(* Logix 5000 project; controller WWTP_SOLIDS_CLX vendor 1 type 14 code 54 rev 17.2; software revision 17.00; part 14 of 16 *)
(* tags used below, declared in another part *)
   Inp_ClosedLS : BOOL;   // Valve Closed Limit Switch 1=confirmed CLOSED
   Inp_OpenPermOK : BOOL;   // 1=Open Permissives OK, Valve can motor open
   Inp_OpenNBPermOK : BOOL;   // 1=Non-Bypassable Open Permissives OK, valve can motor open
   Inp_ClosePermOK : BOOL;   // 1=Close Permissives OK, Valve can motor closed
   Inp_CloseNBPermOK : BOOL;   // 1=Non-Bypassable Close Permissives OK, valve can motor closed
   Inp_IOFault : BOOL;   // Input Communication Status 0=OK, 1=fail
   Inp_Sim : BOOL;   // 1=Simulate working valve; 0=Open/Close/ Monitor actual valve
   Inp_Hand : BOOL;   // 1=Select Hand (hardwired) Mode
   Inp_Reset : BOOL;   // 1=Reset all fault conditions and latched Alarms
   Cfg_HasOpenLS : BOOL;   // 1=Valve provides an Open Limit Switch signal
   Cfg_HasClosedLS : BOOL;   // 1=Valve provides a Closed Limit Switch signal
   Cfg_UseOpenLS : BOOL;   // 1=Valve Open LS should be used for failure checking
   Cfg_UseClosedLS : BOOL;   // 1=Valve Closed LS should be used for failure checking
   Cfg_LSFail : BOOL;   // 1=both switches ON=fail, 0=both switches OFF=fail
   Cfg_HasOpenPermObj : BOOL;   // 1=Tells HMI a P_Perm is connected to Inp_OpenPermOK
   Cfg_HasClosePermObj : BOOL;   // 1=Tells HMI a P_Perm is connected to Inp_ClosePermOK
   Cfg_PCmdClear : BOOL;   // 1=Clear Program Commands on receipt 0=Leave Set
   Cfg_HasFullStallAlm : BOOL;   // 1=Full Stall Alarm exists and will be checked
   Cfg_HasTransitStallAlm : BOOL;   // 1=Transit Stall Alarm exists and will be checked
   Cfg_HasActuatorFaultAlm : BOOL;   // 1=Actuator Fault Alarm exists and will be checked
   Cfg_HasIOFaultAlm : BOOL;   // 1=I/O Fault Alarm exists and will be checked
   Cfg_FullStallAckReqd : BOOL;   // 1=Acknowledge required for Full Stall Alarm
   Cfg_TransitStallAckReqd : BOOL;   // 1=Acknowledge required for Transit Stall Alarm
   Cfg_ActuatorFaultAckReqd : BOOL;   // 1=Acknowledge required for Actuator Fault Alarm
   Cfg_IOFaultAckReqd : BOOL;   // 1=Acknowledge required for I/O Fault Alarm
   Cfg_FullStallSeverity : SINT;   // Full Stall Alarm Severity 1=info 2=warn 3=excep 4=fault
   Cfg_TransitStallSeverity : SINT;   // Transit Stall Alarm Severity 1=info 2=warn 3=excep 4=fault
   Cfg_ActuatorFaultSeverity : SINT;   // Actuator Fault Alarm Severity 1=info 2=warn 3=excep 4=fault
   Cfg_IOFaultSeverity : SINT;   // I/O Fault Alarm Severity 1=info 2=warn 3=excep 4=fault
   Cfg_OutPulseT : DINT;   // Time (in seconds) to pulse valve outputs (0 = outputs maintained ON)
   Cfg_SimFdbkT : DINT;   // Delay to echo back of Open/Closed status when in Simulation (sec)
   Cfg_FullStallT : DINT;   // After commanded, time with no motion before Fault (sec)
   Cfg_TransitStallT : DINT;   // After command, time to reach position before fault (sec)
   PSet_Owner : DINT;   // Program Owner Request ID (non-zero) or Release (zero)
   PCmd_Open : BOOL;   // Program Command to Open Valve
   PCmd_Close : BOOL;   // Program Command to Close Valve
   PCmd_Acq : BOOL;   // Program Command to Acquire ownership (Oper/OOS to Prog)
   PCmd_Rel : BOOL;   // Program Command to Release ownership (Prog to OOS)
   PCmd_Lock : BOOL;   // Program Command to Lock Mode in Prog
   PCmd_Unlock : BOOL;   // Program Command to Unlock Mode
   PCmd_Reset : BOOL;   // Program Command to Reset all Alarms requiring Reset
   PCmd_FullStallInhibit : BOOL;   // Program Command to Inhibit Full Stall Alarm
   PCmd_FullStallUninhibit : BOOL;   // Program Command to Uninhibit Full Stall Alarm
   PCmd_TransitStallInhibit : BOOL;   // Program Command to Inhibit Transit Stall Alarm
   PCmd_TransitStallUninhibit : BOOL;   // Program Command to Uninhibit Transit Stall Alarm
   PCmd_ActuatorFaultInhibit : BOOL;   // Program Command to Inhibit Actuator Fault Alarm
   PCmd_ActuatorFaultUninhibit : BOOL;   // Program Command to Uninhibit Actuator Fault Alarm
   PCmd_IOFaultInhibit : BOOL;   // Program Command to Inhibit I/O Fault Alarm
   PCmd_IOFaultUninhibit : BOOL;   // Program Command to Uninhibit I/O Fault Alarm
   OCmd_Open : BOOL;   // Operator Command to Open Valve
   OCmd_Close : BOOL;   // Operator Command to Close Valve
   OCmd_Stop : BOOL;   // Operator Command to Stop Valve Motion
   OCmd_Bypass : BOOL;   // Operator Command to Bypass all Bypassable Interlocks and Permissives
   OCmd_Check : BOOL;   // Operator Command to Check (not bypass) all Interlocks and Permissives
   MCmd_Disable : BOOL;   // Maintenance Command to Disable Valve
   MCmd_Enable : BOOL;   // Maintenance Command to Enable (allow to energize) Valve
   OCmd_Reset : BOOL;   // Operator Command to Reset all Alarms requiring Reset
   Val_Owner : DINT;   // Current Object Owner ID (0=not owned)
   Val_Notify : SINT;   // Current Alarm Level and Acknowledgement (enumeration)
   Sts_Stopped : BOOL;   // 1=Valve requested to Stop and is not at either end of travel
   Sts_Hand : BOOL;   // 1=Mode is Hand (supersedes Maint, Ovrd, Prog, Oper)
   Sts_Maint : BOOL;   // 1=Mode is Maintenance (supersedes Ovrd, Prog, Oper)
   Sts_Oper : BOOL;   // 1=Mode is Operator (manual)
   Sts_ProgOperLock : BOOL;   // 1=Program or Operator has requested Mode Lock
   Ack_FullStall : BOOL;   // 1=Full Stall Alarm has been acknowledged
   Ack_TransitStall : BOOL;   // 1=Transit Stall Alarm has been acknowledged
   Ack_ActuatorFault : BOOL;   // 1=Actuator Fault Alarm has been acknowledged
   Ack_IOFault : BOOL;   // 1=I/O Fault Alarm has been acknowledged
   Rdy_Open : BOOL;   // 1=Ready to receive OCmd_Open (enables HMI button)
   Rdy_Close : BOOL;   // 1=Ready to receive OCmd_Close (enables HMI button)
   Rdy_Bypass : BOOL;   // 1=Ready to receive OCmd_Bypass (enables HMI button)
   Rdy_Disable : BOOL;   // 1=Ready to receive MCmd_Disable (enables HMI button)
   Rdy_Reset : BOOL;   // 1=Ready to receive OCmd_Reset (enables HMI button)
   Mode : P_Mode;   // Valve Mode Selection
   Wrk_Open : BOOL;   // 1=Requested to OPEN Valve
   Wrk_Stop : BOOL;   // 1=Requested to STOP Valve
   Wrk_Close : BOOL;   // 1-Requested to CLOSE Valve
(* P_ValveMO, continued *)

ROUTINE Prescan   (* ladder *)
// Clear Ownership, set to De-Energized state, clear "lurking" Commands
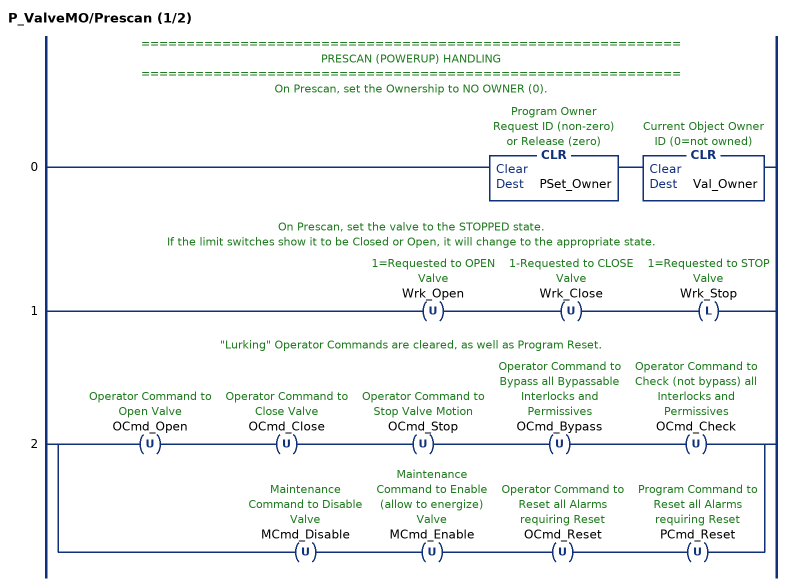
   // ============================================================
   // PRESCAN (POWERUP) HANDLING
   // ============================================================
   // On Prescan, set the Ownership to NO OWNER (0).
   0: CLR(PSet_Owner)CLR(Val_Owner);
   // On Prescan, set the valve to the STOPPED state.
   // If the limit switches show it to be Closed or Open, it will change to the appropriate state.
   1: OTU(Wrk_Open)OTU(Wrk_Close)OTL(Wrk_Stop);
   // "Lurking" Operator Commands are cleared, as well as Program Reset.
   2: [OTU(OCmd_Open) OTU(OCmd_Close) OTU(OCmd_Stop) OTU(OCmd_Bypass) OTU(OCmd_Check) ,OTU(MCmd_Disable) OTU(MCmd_Enable) OTU(OCmd_Reset) OTU(PCmd_Reset) ];
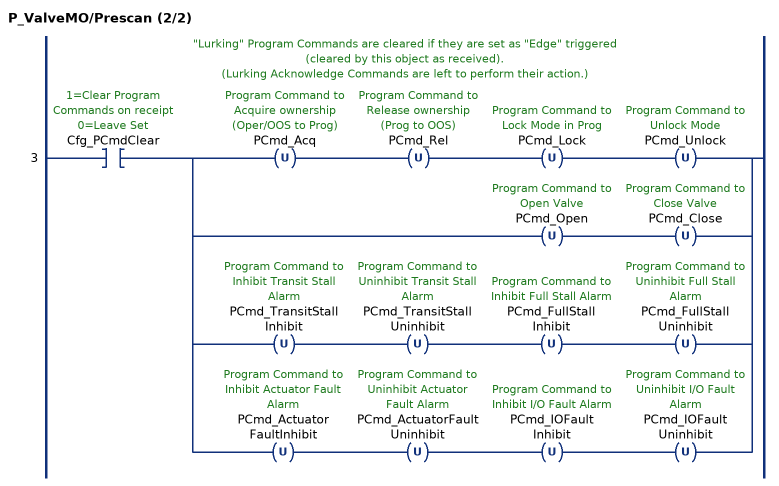
   // "Lurking" Program Commands are cleared if they are set as "Edge" triggered
   // (cleared by this object as received).
   // (Lurking Acknowledge Commands are left to perform their action.)
   3: XIC(Cfg_PCmdClear)[OTU(PCmd_Acq) OTU(PCmd_Rel) OTU(PCmd_Lock) OTU(PCmd_Unlock) ,OTU(PCmd_Open) OTU(PCmd_Close) ,OTU(PCmd_TransitStallInhibit) OTU(PCmd_TransitStallUninhibit) OTU(PCmd_FullStallInhibit) OTU(PCmd_FullStallUninhibit) ,OTU(PCmd_ActuatorFaultInhibit) OTU(PCmd_ActuatorFaultUninhibit) OTU(PCmd_IOFaultInhibit) OTU(PCmd_IOFaultUninhibit) ];
END_ROUTINE
END_ADD_ON_INSTRUCTION

ADD_ON_INSTRUCTION U_CommFail   (* revision 1.0 *)
// Communication Failure Between two PLCs
VAR_INPUT
   Inp_Heartbeat : BOOL; {visible}   // Heartbeat from Remote PLC
   CFG_DelayTimerSec : DINT := 30; {visible}   // Delay Timer in Seconds
END_VAR
VAR_OUTPUT
   Sts_CommFail : BOOL; {visible}   // Communication Failure Alarm
END_VAR
VAR
   HeartBeatDelayTimerOn : TIMER;
   HeartBeatDelayTimerOff : TIMER;
   ConnectionStatusDelayTimer : TIMER;
END_VAR

ROUTINE Logic   (* ladder *)
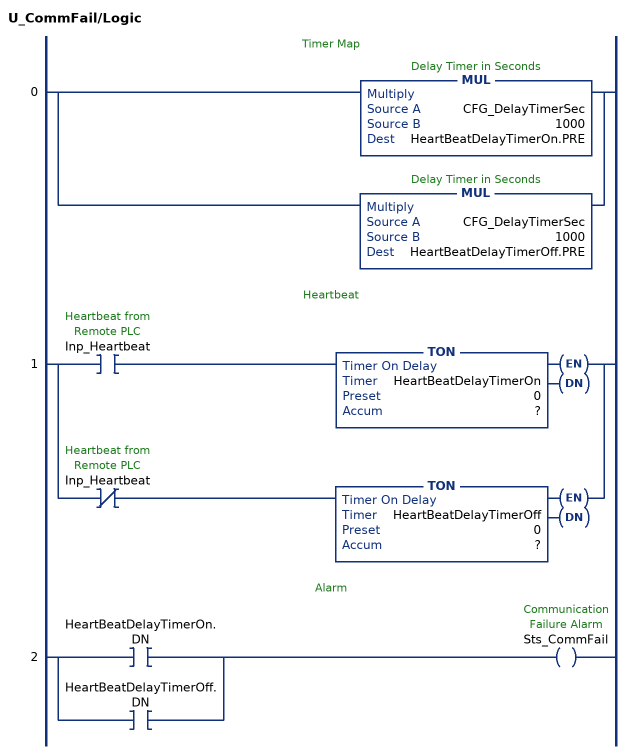
   // Timer Map
   0: [MUL(CFG_DelayTimerSec,1000,HeartBeatDelayTimerOn.PRE) ,MUL(CFG_DelayTimerSec,1000,HeartBeatDelayTimerOff.PRE) ];
   // Heartbeat
   1: [XIC(Inp_Heartbeat) TON(HeartBeatDelayTimerOn,?,?) ,XIO(Inp_Heartbeat) TON(HeartBeatDelayTimerOff,?,?) ];
   // Alarm
   2: [XIC(HeartBeatDelayTimerOn.DN) ,XIC(HeartBeatDelayTimerOff.DN) ]OTE(Sts_CommFail);
END_ROUTINE
END_ADD_ON_INSTRUCTION

ADD_ON_INSTRUCTION U_FlowTot   (* revision 1.0 *)
// Provides Totalization for Daily & Yearly Flow.
VAR_IN_OUT
   Inp_AIn : P_AIn; {required}   // Flow Analog Input AOI
   Inp_WallClock : U_WallClock; {required}   // PLC Wall Clock
END_VAR
VAR_INPUT
   Inp_ProgStartReq : BOOL := 1;   // Prog Start Request. If needed map to turn on totalizer, (ex. pump running) else Defaults to 1 (always start)
END_VAR
VAR_OUTPUT
   Val_FlowRate : REAL; {visible}   // Current Flow Rate
   Val_DailyTot : REAL; {visible}   // Todays Total Flow
   Val_YestTot : REAL; {visible}   // Yesterday Total Flow
   Val_YearlyTot : REAL; {visible}   // This Year Total Flow
   Val_LastYearTot : REAL; {visible}   // Last Year Total Flow
END_VAR
VAR
   YearlyTotalizer : TOTALIZER := (TimeBase := 3, Gain := 1.0, ProgProgReq := 1, ProgStartReq := 1, OperStartReq := 1, RTSTime := 1, ProgOper := 1, RunStop := 1, TargetFlag := 1, TargetDev1Flag := 1, TargetDev2Flag := 1, DeltaT := 0.010000001);
   DailyTotalizer : TOTALIZER := (TimeBase := 3, Gain := 100000.0, ProgStartReq := 1, OperStartReq := 1, RTSTime := 1, ProgOper := 1, RunStop := 1, TargetFlag := 1, TargetDev1Flag := 1, TargetDev2Flag := 1, DeltaT := 0.010000001);
   FlowRateLowLimit_SSUM : SELECTED_SUMMER := (Gain1 := 1.0, Gain2 := 1.0, Gain3 := 1.0, Gain4 := 1.0, Gain5 := 1.0, Gain6 := 1.0, Gain7 := 1.0, Gain8 := 1.0);
   LowCutoff_BNOT : FBD_BOOLEAN_NOT := (In := 1);
   __l00009BB0 : DINT;
   __l00004A73 : REAL;
   __l0000B40A : BOOL;
   __l000041A5 : DINT;
END_VAR

ROUTINE Logic   (* function block diagram *)
   SHEET 1   // Main
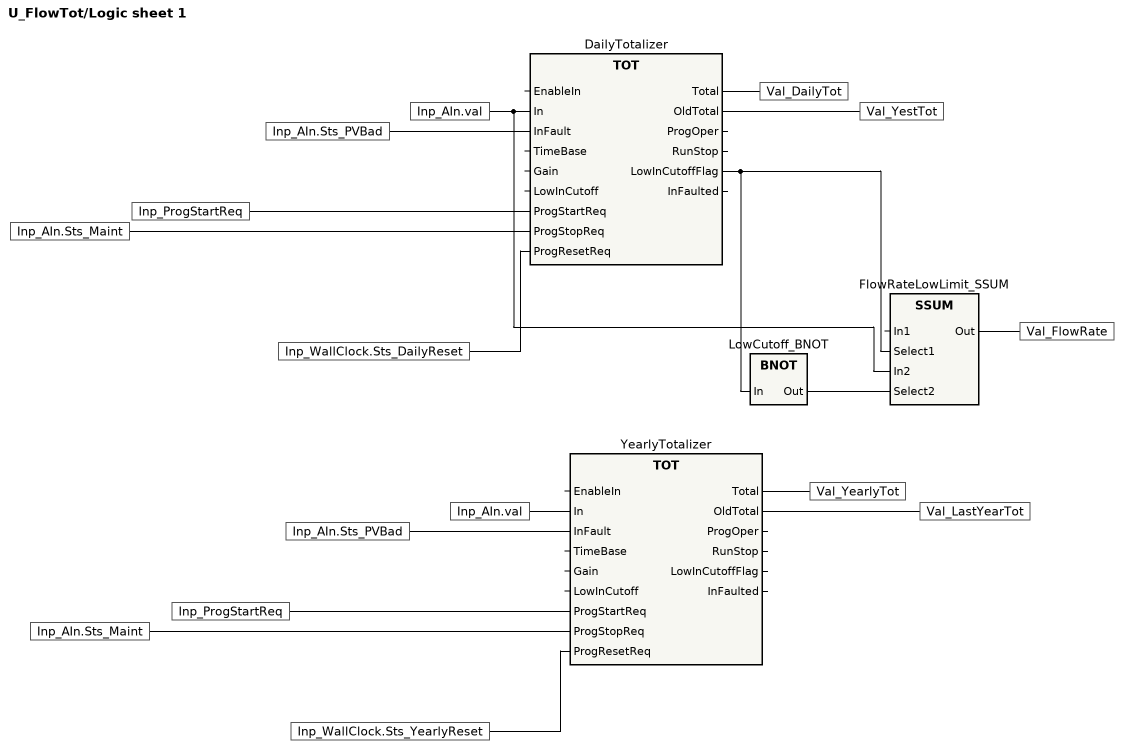
   DailyTotalizer : TOT(In := Inp_AIn.val, InFault := Inp_AIn.Sts_PVBad, ProgStartReq := Inp_ProgStartReq, ProgStopReq := Inp_AIn.Sts_Maint, ProgResetReq := Inp_WallClock.Sts_DailyReset);   // unwired pins: EnableIn TimeBase Gain LowInCutoff ProgOper RunStop InFaulted
   YearlyTotalizer : TOT(In := Inp_AIn.val, InFault := Inp_AIn.Sts_PVBad, ProgStartReq := Inp_ProgStartReq, ProgStopReq := Inp_AIn.Sts_Maint, ProgResetReq := Inp_WallClock.Sts_YearlyReset);   // unwired pins: EnableIn TimeBase Gain LowInCutoff ProgOper RunStop LowInCutoffFlag InFaulted
   LowCutoff_BNOT : BNOT(In := DailyTotalizer.LowInCutoffFlag);
   Val_DailyTot := DailyTotalizer.Total;
   Val_YearlyTot := YearlyTotalizer.Total;
   Val_YestTot := DailyTotalizer.OldTotal;
   FlowRateLowLimit_SSUM : SSUM(Select1 := DailyTotalizer.LowInCutoffFlag, In2 := Inp_AIn.val, Select2 := LowCutoff_BNOT.Out);   // unwired pins: In1
   Val_LastYearTot := YearlyTotalizer.OldTotal;
   Val_FlowRate := FlowRateLowLimit_SSUM.Out;
END_ROUTINE
END_ADD_ON_INSTRUCTION

ADD_ON_INSTRUCTION U_Heartbeat   (* revision 1.0 *)
// Heartbeat Between two PLCs
VAR_INPUT
   CFG_DelayTimerSec : DINT := 30; {visible}   // Delay Timer in Seconds
END_VAR
VAR_OUTPUT
   Heartbeat : BOOL; {visible}   // Heartbeat from Remote PLC
END_VAR
VAR
   DelayTimerOn : TIMER;
   DelayTimerOff : TIMER;
END_VAR

ROUTINE Logic   (* ladder *)
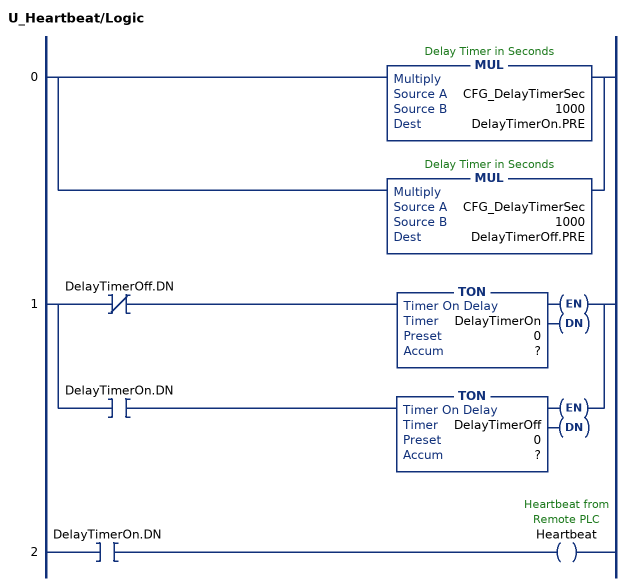
   0: [MUL(CFG_DelayTimerSec,1000,DelayTimerOn.PRE) ,MUL(CFG_DelayTimerSec,1000,DelayTimerOff.PRE) ];
   1: [XIO(DelayTimerOff.DN) TON(DelayTimerOn,?,?) ,XIC(DelayTimerOn.DN) TON(DelayTimerOff,?,?) ];
   2: XIC(DelayTimerOn.DN)OTE(Heartbeat);
END_ROUTINE
END_ADD_ON_INSTRUCTION

ADD_ON_INSTRUCTION U_WallClock   (* revision 1.1 *)
// Wall Clock Set time, Current time and Reset bits.
// Revision note:
// Simplified Day of Week calculation, removed unused tags as a result.
VAR_INPUT
   OCmd_SetTime : BOOL; {visible}   // Set the Date and Time Bit
   OSet_Year : DINT; {visible}   // Year To Set
   OSet_Month : DINT; {visible}   // Month To Set
   OSet_Day : DINT; {visible}   // Day To Set
   OSet_Hour : DINT; {visible}   // Hour To Set
   OSet_Minute : DINT; {visible}   // Minute To Set
   OSet_Second : DINT; {visible}   // Second To Set
END_VAR
VAR_OUTPUT
   Val_CurrentYear : DINT; {visible}   // Current Year
   Val_CurrentMonth : DINT; {visible}   // Current Month
   Val_CurrentDay : DINT; {visible}   // Current Day
   Val_CurrentHour : DINT; {visible}   // Current Hour
   Val_CurrentMinute : DINT; {visible}   // Current Minute
   Val_CurrentSecond : DINT; {visible}   // Current Second
   Val_DayOfWeek : DINT; {visible}   // Day of Week 0 = Sun, 1=Mon, 2=Tues, 3=Wed, 4=Thur, 5=Fri, 6=Sat
   Sts_HourlyReset : BOOL; {visible}   // Hourly Reset
   Sts_DailyReset : BOOL; {visible}   // Daily Reset
   Sts_MonthlyReset : BOOL; {visible}   // Monthly Reset
   Sts_YearlyReset : BOOL; {visible}   // Yearly Reset
END_VAR
VAR
   Wrk_SetDateTime : DINT[7];
   Wrk_GetDateTime : DINT[7];   // Result of GSV to Wallclocktime -- input to Day of Week calculation
        [0]   // Year
        [1]   // Month
        [2]   // Day
        [3]   // Hour
        [4]   // Minute
        [5]   // Second
        [6]   // Microsecond
   Wrk_G : DINT;   // Function of Year and Month, used to calculate Day of Week
   Wrk_F : DINT;   // Function of Month, used to calculate Day of Week
   Wrk_DayONS : BOOL;   // One-Shot for daily pulse output
   Wrk_HourONS : BOOL;   // One-Shot for hourly pulse output
   Wrk_MonthONS : BOOL;   // One-Shot for monthly pulse output
   Wrk_YearONS : BOOL;   // One-Shot for yearly pulse output
END_VAR

ROUTINE Logic   (* ladder *)
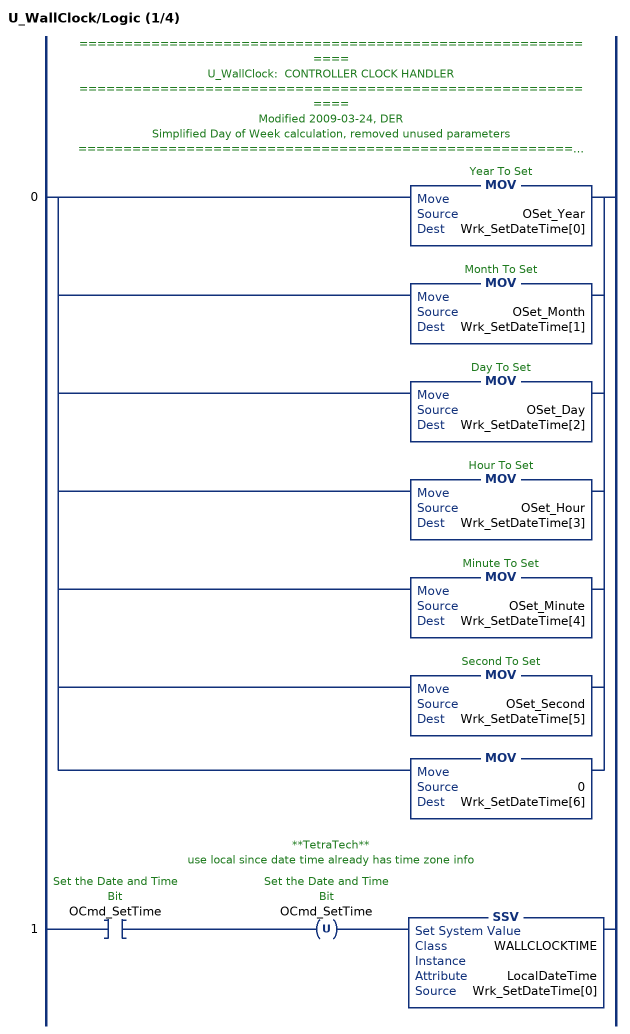
   // ============================================================
   // U_WallClock:  CONTROLLER CLOCK HANDLER
   // ============================================================
   // Modified 2009-03-24, DER
   // Simplified Day of Week calculation, removed unused parameters
   // ============================================================
   // This object manages the controller "Wall Clock", providing date and time services
   // including:
   // * Accepts downloaded date and time and "Set" command from HMI or other sync source and sets the clock
   // * Reads the clock and provides the local date and time to other logic
   // * Calculates and provides the day of the week for the current date
   // * Sets a flag every Hour, Day, Month and Year for resets / data collectors
   // The time is provided as separate Values:
   // Val_CurrentYear : DINT,
   // Val_CurrentMonth : DINT,
   // Val_CurrentDay : DINT,
   // Val_CurrentHour : DINT,
   // Val_CurrentMinute : DINT,
   // Val_CurrentSecond : DINT,
   // Val_DayOfWeek : DINT)
   // ============================================================
   // HANDLE RECEIVED DATE/TIME SYNC, SET CLOCK
   // ============================================================
   // If a date and time have been received with a "Set" command,
   // store the date/time to the controller clock.
   0: [MOV(OSet_Year,Wrk_SetDateTime[0]) ,MOV(OSet_Month,Wrk_SetDateTime[1]) ,MOV(OSet_Day,Wrk_SetDateTime[2]) ,MOV(OSet_Hour,Wrk_SetDateTime[3]) ,MOV(OSet_Minute,Wrk_SetDateTime[4]) ,MOV(OSet_Second,Wrk_SetDateTime[5]) ,MOV(0,Wrk_SetDateTime[6]) ];
   // **TetraTech**
   // use local since date time already has time zone info
   1: XIC(OCmd_SetTime)OTU(OCmd_SetTime)SSV(WALLCLOCKTIME,,LocalDateTime,Wrk_SetDateTime[0]);
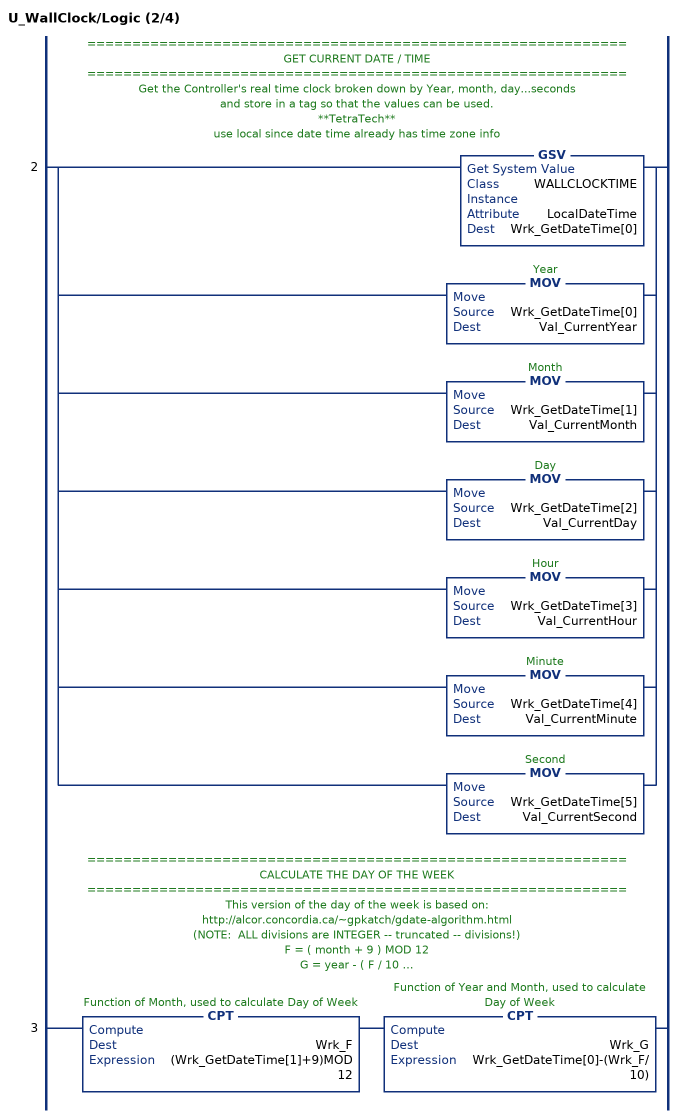
   // ============================================================
   // GET CURRENT DATE / TIME
   // ============================================================
   // Get the Controller's real time clock broken down by Year, month, day...seconds
   // and store in a tag so that the values can be used.
   // **TetraTech**
   // use local since date time already has time zone info
   2: [GSV(WALLCLOCKTIME,,LocalDateTime,Wrk_GetDateTime[0]) ,MOV(Wrk_GetDateTime[0],Val_CurrentYear) ,MOV(Wrk_GetDateTime[1],Val_CurrentMonth) ,MOV(Wrk_GetDateTime[2],Val_CurrentDay) ,MOV(Wrk_GetDateTime[3],Val_CurrentHour) ,MOV(Wrk_GetDateTime[4],Val_CurrentMinute) ,MOV(Wrk_GetDateTime[5],Val_CurrentSecond) ];
   // ============================================================
   // CALCULATE THE DAY OF THE WEEK
   // ============================================================
   // This version of the day of the week is based on:
   // http://alcor.concordia.ca/~gpkatch/gdate-algorithm.html
   // (NOTE:  ALL divisions are INTEGER -- truncated -- divisions!)
   // F = ( month + 9 ) MOD 12
   // G = year - ( F / 10 )
   // Gregorian DayNumber [ D ] = ( 365 * G ) + ( G / 4 ) - ( G / 100 ) + ( G / 400 ) + ( ( ( F * 306 ) + 5 ) / 10 ) + day - 1
   // DayOfWeek = ( DayNumber + 3 ) MOD 7
   // ~~~~~~~~~~~~~~~~~~~~~~~~~~~~~~~~~~~~~~~~~~~~~~~~~~~~~~~~~~~~
   // This rung calculates the "G" and "F" functions shown in the algorithm above.
   // ~~~~~~~~~~~~~~~~~~~~~~~~~~~~~~~~~~~~~~~~~~~~~~~~~~~~~~~~~~~~
   3: CPT(Wrk_F,(Wrk_GetDateTime[1]+9)MOD 12)CPT(Wrk_G,Wrk_GetDateTime[0]-(Wrk_F/10));
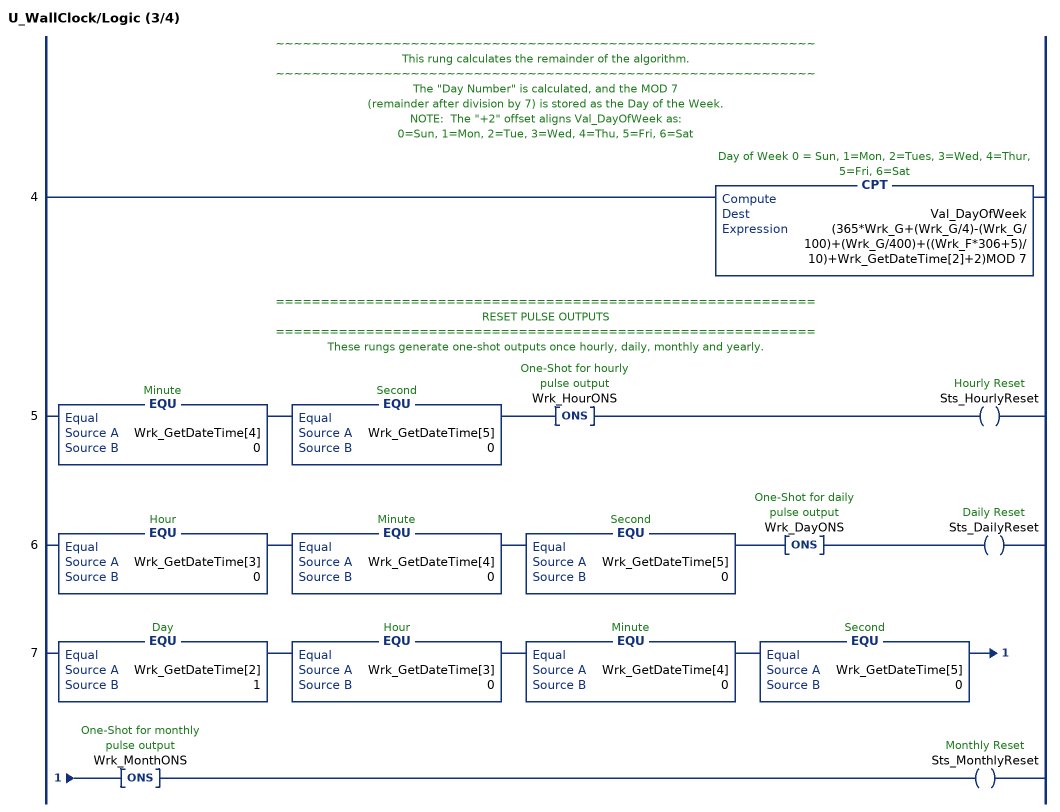
   // ~~~~~~~~~~~~~~~~~~~~~~~~~~~~~~~~~~~~~~~~~~~~~~~~~~~~~~~~~~~~
   // This rung calculates the remainder of the algorithm.
   // ~~~~~~~~~~~~~~~~~~~~~~~~~~~~~~~~~~~~~~~~~~~~~~~~~~~~~~~~~~~~
   // The "Day Number" is calculated, and the MOD 7
   // (remainder after division by 7) is stored as the Day of the Week.
   // NOTE:  The "+2" offset aligns Val_DayOfWeek as:
   // 0=Sun, 1=Mon, 2=Tue, 3=Wed, 4=Thu, 5=Fri, 6=Sat
   4: CPT(Val_DayOfWeek,(365*Wrk_G+(Wrk_G/4)-(Wrk_G/100)+(Wrk_G/400)+((Wrk_F*306+5)/10)+Wrk_GetDateTime[2]+2)MOD 7);
   // ============================================================
   // RESET PULSE OUTPUTS
   // ============================================================
   // These rungs generate one-shot outputs once hourly, daily, monthly and yearly.
   5: EQU(Wrk_GetDateTime[4],0)EQU(Wrk_GetDateTime[5],0)ONS(Wrk_HourONS)OTE(Sts_HourlyReset);
   6: EQU(Wrk_GetDateTime[3],0)EQU(Wrk_GetDateTime[4],0)EQU(Wrk_GetDateTime[5],0)ONS(Wrk_DayONS)OTE(Sts_DailyReset);
   7: EQU(Wrk_GetDateTime[2],1)EQU(Wrk_GetDateTime[3],0)EQU(Wrk_GetDateTime[4],0)EQU(Wrk_GetDateTime[5],0)ONS(Wrk_MonthONS)OTE(Sts_MonthlyReset);
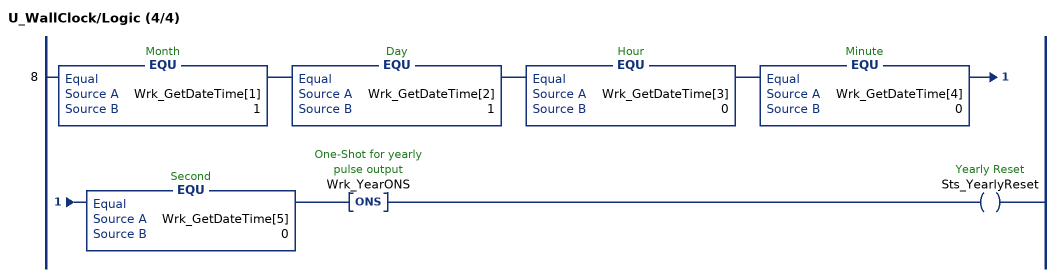
   8: EQU(Wrk_GetDateTime[1],1)EQU(Wrk_GetDateTime[2],1)EQU(Wrk_GetDateTime[3],0)EQU(Wrk_GetDateTime[4],0)EQU(Wrk_GetDateTime[5],0)ONS(Wrk_YearONS)OTE(Sts_YearlyReset);
END_ROUTINE
END_ADD_ON_INSTRUCTION

VAR_GLOBAL   (* controller tags *)
   I_P600_Fault : ALIAS FOR Local:3:I.DATA.1;
   I_P600_Fault_IOFault : ALIAS FOR Local:3:I.Fault.1;
   I_P600_InAuto : ALIAS FOR Local:3:I.Data.4;
   I_P600_InAuto_IOFault : ALIAS FOR Local:3:I.Fault.4;
   I_P600_RunFdbk : ALIAS FOR Local:3:I.Data.2;
   I_P600_RunFdbk_IOFault : ALIAS FOR Local:3:I.Fault.2;
   I_P601_Fault : ALIAS FOR Local:3:I.Data.6;
   I_P601_Fault_IOFault : ALIAS FOR Local:3:I.Fault.6;
   I_P601_InAuto : ALIAS FOR Local:3:I.Data.4;
   I_P601_InAuto_IOFault : ALIAS FOR Local:3:I.Fault.4;
   I_P601_RunFdbk : ALIAS FOR Local:3:I.Data.5;
   I_P601_RunFdbk_IOFault : ALIAS FOR Local:3:I.Fault.5;
   I_P602_Fault : ALIAS FOR Local:3:I.Data.9;
   I_P602_Fault_IOFault : ALIAS FOR Local:3:I.Fault.9;
   I_P602_InAuto : ALIAS FOR Local:3:I.Data.7;
   I_P602_InAuto_IOFault : ALIAS FOR Local:3:I.Fault.7;
   I_P602_RunFdbk : ALIAS FOR Local:3:I.Data.8;
   I_P602_RunFdbk_IOFault : ALIAS FOR Local:3:I.Fault.8;
   I_PV600_CloseLS : ALIAS FOR Local:3:I.Data.14;
   I_PV600_CloseLS_IOFault : ALIAS FOR Local:3:I.Fault.14;
   I_PV600_InAuto : ALIAS FOR Local:3:I.Data.0;
   I_PV600_InAuto_IOFault : ALIAS FOR Local:3:I.Fault.0;
   I_PV600_OpenLS : ALIAS FOR Local:3:I.Data.13;
   I_PV600_OpenLS_IOFault : ALIAS FOR Local:3:I.Fault.13;
   I_SecRAS_ToGBT_Flow : ALIAS FOR Local:5:I.CH0DATA;
   I_SecRAS_ToGBT_Flow_IOFault : ALIAS FOR Local:5:I.CH0Fault;
   I_SolidsTk_Lv : ALIAS FOR Local:5:I.Ch1Data;
   I_SolidsTk_Lv_IOFault : ALIAS FOR Local:5:I.Ch1Fault;
   I_SolidsTkDrive_InAuto : ALIAS FOR Local:3:I.Data.10;
   I_SolidsTkDrive_InAuto_IOFault : ALIAS FOR Local:3:I.Fault.10;
   I_SolidsTkDrive_RunFdbk : ALIAS FOR Local:3:I.Data.11;
   I_SolidsTkDrive_RunFdbk_IOFault : ALIAS FOR Local:3:I.Fault.11;
   I_SolidsTkDrive_Torque : ALIAS FOR Local:3:I.Data.12;
   I_SolidsTkDrive_Torque_IOFault : ALIAS FOR Local:3:I.Fault.12;
   I_WAS_HoldTkLv : ALIAS FOR Local:5:I.Ch3Data;
   I_WAS_HoldTkLv_IOFault : ALIAS FOR Local:5:I.Ch3Fault;
   I_WAS_StorageTk_Lv : ALIAS FOR Local:5:I.Ch2Data;
   I_WAS_StorageTk_Lv_IOFault : ALIAS FOR Local:5:I.Ch2Fault;
   O_P600_Out_Run : ALIAS FOR Local:4:O.Data.1;   // P-600 Start/Stop
   O_P601_Out_Run : ALIAS FOR Local:4:O.Data.2;   // P-601 Start/Stop
   O_P602_Out_Run : ALIAS FOR Local:4:O.Data.3;   // P-602 Start/Stop
   O_PV600_Close : ALIAS FOR Local:4:O.Data.5;   // P-600 Close
   O_PV600_Open : ALIAS FOR Local:4:O.Data.4;   // P-600 Open
   O_SolidsTkDrive_Out_Run : ALIAS FOR Local:4:O.DATA.0;   // Solids Storage Tank #1 Drive Start/Stop
   P600_Fault : P_DIn := (Inp_Gate := 1, Cfg_NormTextVis := 1, Cfg_PCmdClear := 1, Cfg_TgtDisagreeAckReqd := 1, Cfg_TgtDisagreeSeverity := 3, Sts_InpPV := 1, Ack_TgtDisagree := 1, Rdy_SubstPV := 1);   // P-600 Fault
   P600_Intlk : P_Intlk := (Cfg_PCmdClear := 1, Sts_IntlkOK := 1, Sts_NBIntlkOK := 1);   // P-600 Interlock
   P600_Motor : P_Motor := (Inp_PermOK := 1, Inp_NBPermOK := 1, Inp_IntlkOK := 1, Inp_NBIntlkOK := 1, Inp_Sim := 1, Inp_Hand := 1, Cfg_FailToStartAckReqd := 1, Cfg_FailToStopAckReqd := 1, Cfg_IntlkTripAckReqd := 1, Cfg_IOFaultAckReqd := 1, Cfg_FailToStartSeverity := 4, Cfg_FailToStopSeverity := 4, Cfg_IntlkTripSeverity := 2, Cfg_IOFaultSeverity := 4, Cfg_SimFdbkT := 2, Cfg_FailToStartT := 10, Cfg_FailToStopT := 10, PCmd_Acq := 1, Sts_Hand := 1, Ack_FailToStart := 1, Ack_FailToStop := 1, Ack_IntlkTrip := 1, Ack_IOFault := 1, Rdy_Bypass := 1, Rdy_Disable := 1);   // P-600 Motor
   P600_Perm : P_Perm := (Inp_Perm00 := 1, Inp_Perm01 := 1, Inp_Perm02 := 1, Inp_Perm03 := 1, Inp_Perm04 := 1, Inp_Perm05 := 1, Inp_Perm06 := 1, Inp_Perm07 := 1, Inp_Perm08 := 1, Inp_Perm09 := 1, Inp_Perm10 := 1, Inp_Perm11 := 1, Inp_Perm12 := 1, Inp_Perm13 := 1, Inp_Perm14 := 1, Inp_Perm15 := 1, Sts_PermOK := 1, Sts_NBPermOK := 1, Sts_Perm := 2#1111_1111_1111_1111);   // P-600 Permissive
   P600_Reset : P_Reset := (Cfg_MinHoldTime := 1);   // P-600 Reset
   P600_ResInh : P_ResInh := (Cfg_ThreeColdStarts := 1800, Cfg_FirstFailCold := 1800, Cfg_SubseqFailCold := 14400, Cfg_FirstFailHot := 1800, Cfg_SubseqFailHot := 14400, Cfg_HotRestartOK := 3600, Cfg_RestartHot := 3600, Cfg_HotToCold := 57600, Val_State := 1, Sts_Ready := 1);   // P-600 Restart Inhibit
   P600_RunTime : P_RunTime := (Cfg_PCmdClear := 1);   // P-600 Run Time
   P601_Fault : P_DIn := (Inp_Gate := 1, Cfg_NormTextVis := 1, Cfg_PCmdClear := 1, Cfg_TgtDisagreeAckReqd := 1, Cfg_TgtDisagreeSeverity := 3, Sts_InpPV := 1, Ack_TgtDisagree := 1, Rdy_SubstPV := 1);   // P-601 Fault
   P601_Intlk : P_Intlk := (Cfg_PCmdClear := 1, Sts_IntlkOK := 1, Sts_NBIntlkOK := 1);   // P-601 Interlock
   P601_Motor : P_Motor := (Inp_PermOK := 1, Inp_NBPermOK := 1, Inp_IntlkOK := 1, Inp_NBIntlkOK := 1, Inp_Sim := 1, Inp_Hand := 1, Cfg_FailToStartAckReqd := 1, Cfg_FailToStopAckReqd := 1, Cfg_IntlkTripAckReqd := 1, Cfg_IOFaultAckReqd := 1, Cfg_FailToStartSeverity := 4, Cfg_FailToStopSeverity := 4, Cfg_IntlkTripSeverity := 2, Cfg_IOFaultSeverity := 4, Cfg_SimFdbkT := 2, Cfg_FailToStartT := 10, Cfg_FailToStopT := 10, PCmd_Acq := 1, Sts_Hand := 1, Ack_FailToStart := 1, Ack_FailToStop := 1, Ack_IntlkTrip := 1, Ack_IOFault := 1, Rdy_Bypass := 1, Rdy_Disable := 1);   // P-601 Motor
   P601_Perm : P_Perm := (Inp_Perm00 := 1, Inp_Perm01 := 1, Inp_Perm02 := 1, Inp_Perm03 := 1, Inp_Perm04 := 1, Inp_Perm05 := 1, Inp_Perm06 := 1, Inp_Perm07 := 1, Inp_Perm08 := 1, Inp_Perm09 := 1, Inp_Perm10 := 1, Inp_Perm11 := 1, Inp_Perm12 := 1, Inp_Perm13 := 1, Inp_Perm14 := 1, Inp_Perm15 := 1, Sts_PermOK := 1, Sts_NBPermOK := 1, Sts_Perm := 2#1111_1111_1111_1111);   // P-601 Permissive
   P601_Reset : P_Reset := (Cfg_MinHoldTime := 1);   // P-601 Reset
   P601_ResInh : P_ResInh := (Cfg_ThreeColdStarts := 1800, Cfg_FirstFailCold := 1800, Cfg_SubseqFailCold := 14400, Cfg_FirstFailHot := 1800, Cfg_SubseqFailHot := 14400, Cfg_HotRestartOK := 3600, Cfg_RestartHot := 3600, Cfg_HotToCold := 57600, Val_State := 1, Sts_Ready := 1);   // P-601 Restart Inhibit
   P601_RunTime : P_RunTime := (Cfg_PCmdClear := 1);   // P-601 Run Time
   P602_Fault : P_DIn := (Inp_Gate := 1, Cfg_NormTextVis := 1, Cfg_PCmdClear := 1, Cfg_TgtDisagreeAckReqd := 1, Cfg_TgtDisagreeSeverity := 3, Sts_SubstPV := 1, Ack_TgtDisagree := 1, Rdy_InpPV := 1);   // P-602 Fault
   P602_Intlk : P_Intlk := (Cfg_PCmdClear := 1, Sts_IntlkOK := 1, Sts_NBIntlkOK := 1);   // P-602 Interlock
   P602_Motor : P_Motor := (Inp_PermOK := 1, Inp_NBPermOK := 1, Inp_IntlkOK := 1, Inp_NBIntlkOK := 1, Inp_Sim := 1, Cfg_HasRunFdbk := 1, Cfg_UseRunFdbk := 1, Cfg_HasPermObj := 1, Cfg_HasIntlkObj := 1, Cfg_HasResInhObj := 1, Cfg_HasRunTimeObj := 1, Cfg_HasFailToStartAlm := 1, Cfg_HasFailToStopAlm := 1, Cfg_FailToStartAckReqd := 1, Cfg_FailToStopAckReqd := 1, Cfg_IntlkTripAckReqd := 1, Cfg_IOFaultAckReqd := 1, Cfg_FailToStartSeverity := 4, Cfg_FailToStopSeverity := 4, Cfg_IntlkTripSeverity := 2, Cfg_IOFaultSeverity := 4, Cfg_SimFdbkT := 2, Cfg_FailToStartT := 10, Cfg_FailToStopT := 10, PCmd_Acq := 1, Sts_Stopped := 1, Sts_Oper := 1, Sts_ProgOperLock := 1, Ack_FailToStart := 1, Ack_FailToStop := 1, Ack_IntlkTrip := 1, Ack_IOFault := 1, Rdy_Start := 1, Rdy_Bypass := 1, Rdy_Disable := 1);   // P-602 Motor
   P602_Perm : P_Perm := (Inp_Perm00 := 1, Inp_Perm01 := 1, Inp_Perm02 := 1, Inp_Perm03 := 1, Inp_Perm04 := 1, Inp_Perm05 := 1, Inp_Perm06 := 1, Inp_Perm07 := 1, Inp_Perm08 := 1, Inp_Perm09 := 1, Inp_Perm10 := 1, Inp_Perm11 := 1, Inp_Perm12 := 1, Inp_Perm13 := 1, Inp_Perm14 := 1, Inp_Perm15 := 1, Sts_PermOK := 1, Sts_NBPermOK := 1, Sts_Perm := 2#1111_1111_1111_1111);   // P-602 Permissive
   P602_Reset : P_Reset := (Cfg_MinHoldTime := 1);   // P-602 Reset
   P602_ResInh : P_ResInh := (Inp_Stopped := 1, Cfg_ThreeColdStarts := 1800, Cfg_FirstFailCold := 1800, Cfg_SubseqFailCold := 14400, Cfg_FirstFailHot := 1800, Cfg_SubseqFailHot := 14400, Cfg_HotRestartOK := 3600, Cfg_RestartHot := 3600, Cfg_HotToCold := 57600, Val_State := 1, Sts_Ready := 1);   // P-602 Restart Inhibit
   P602_RunTime : P_RunTime := (Cfg_PCmdClear := 1, Val_Starts := 1, Val_CurRunHrs := 0.0007227778, Val_MaxRunHrs := 0.0007227778);   // P-602 Run Time
   PLC_CommFail : U_CommFail := (Inp_Heartbeat := 1, CFG_DelayTimerSec := 30, Sts_CommFail := 1);
   PLC_Device_ResetPB : BOOL;   // Site Wide Device Reset Push Button
   PLC_Heartbeat : U_Heartbeat := (CFG_DelayTimerSec := 30, Heartbeat := 1);   // PLC Heartbeat
   PLC_Simulation : BOOL := 1;   // Application running IN SIMULATION
   PLC_WallClock : U_WallClock := (Val_CurrentYear := 1998, Val_CurrentMonth := 2, Val_CurrentDay := 23, Val_CurrentHour := 21, Val_CurrentMinute := 39, Val_CurrentSecond := 15, Val_DayOfWeek := 1);   // Wall Clock
   PV600 : P_ValveMO := (Inp_ClosedLS := 1, Inp_OpenPermOK := 1, Inp_OpenNBPermOK := 1, Inp_ClosePermOK := 1, Inp_CloseNBPermOK := 1, Inp_Sim := 1, Cfg_HasOpenLS := 1, Cfg_HasClosedLS := 1, Cfg_UseOpenLS := 1, Cfg_UseClosedLS := 1, Cfg_LSFail := 1, Cfg_HasOpenPermObj := 1, Cfg_HasClosePermObj := 1, Cfg_PCmdClear := 1, Cfg_HasFullStallAlm := 1, Cfg_HasTransitStallAlm := 1, Cfg_HasActuatorFaultAlm := 1, Cfg_HasIOFaultAlm := 1, Cfg_FullStallAckReqd := 1, Cfg_TransitStallAckReqd := 1, Cfg_ActuatorFaultAckReqd := 1, Cfg_IOFaultAckReqd := 1, Cfg_FullStallSeverity := 4, Cfg_TransitStallSeverity := 4, Cfg_ActuatorFaultSeverity := 2, Cfg_IOFaultSeverity := 4, Cfg_OutPulseT := 5, Cfg_SimFdbkT := 20, Cfg_FullStallT := 15, Cfg_TransitStallT := 60, Sts_Stopped := 1, Sts_Oper := 1, Sts_ProgOperLock := 1, Ack_FullStall := 1, Ack_TransitStall := 1, Ack_ActuatorFault := 1, Ack_IOFault := 1, Rdy_Open := 1, Rdy_Close := 1, Rdy_Bypass := 1, Rdy_Disable := 1);   // Thickened WAS Tank Position Valve (PV-600)
   PV600_ClosePerm : P_Perm := (Inp_Perm00 := 1, Inp_Perm01 := 1, Inp_Perm02 := 1, Inp_Perm03 := 1, Inp_Perm04 := 1, Inp_Perm05 := 1, Inp_Perm06 := 1, Inp_Perm07 := 1, Inp_Perm08 := 1, Inp_Perm09 := 1, Inp_Perm10 := 1, Inp_Perm11 := 1, Inp_Perm12 := 1, Inp_Perm13 := 1, Inp_Perm14 := 1, Inp_Perm15 := 1, Sts_PermOK := 1, Sts_NBPermOK := 1, Sts_Perm := 2#1111_1111_1111_1111);   // Thickened WAS Tank Valve (PV-600) Close Permissive
   PV600_OpenPerm : P_Perm := (Inp_Perm00 := 1, Inp_Perm01 := 1, Inp_Perm02 := 1, Inp_Perm03 := 1, Inp_Perm04 := 1, Inp_Perm05 := 1, Inp_Perm06 := 1, Inp_Perm07 := 1, Inp_Perm08 := 1, Inp_Perm09 := 1, Inp_Perm10 := 1, Inp_Perm11 := 1, Inp_Perm12 := 1, Inp_Perm13 := 1, Inp_Perm14 := 1, Inp_Perm15 := 1, Sts_PermOK := 1, Sts_NBPermOK := 1, Sts_Perm := 2#1111_1111_1111_1111);   // Thickened WAS Tank Valve (PV-600) Open Permissive
   PV600_Reset : P_Reset := (Cfg_MinHoldTime := 1);   // Thickened WAS Tank Valve (PV-600) Reset
   SecRAS_ToGBT_Flow_AIn : P_AIn := (Inp_PV := 500.0, Cfg_SetTrack := 1, Cfg_PCmdClear := 1, Cfg_HiHiAckReqd := 1, Cfg_HiAckReqd := 1, Cfg_LoAckReqd := 1, Cfg_LoLoAckReqd := 1, Cfg_FailAckReqd := 1, Cfg_HiHiSeverity := 3, Cfg_HiSeverity := 2, Cfg_LoSeverity := 2, Cfg_LoLoSeverity := 3, Cfg_FailSeverity := 4, Cfg_InpRawMax := 20.0, Cfg_PVEUMax := 20.0, Cfg_HiHiDB := 1.0, Cfg_HiDB := 1.0, Cfg_LoDB := 1.0, Cfg_LoLoDB := 1.0, Cfg_FailHiLim := 21.0, Cfg_FailLoLim := -1.0, PSet_HiHiLim := 1.5e+38, PSet_HiLim := 1.5e+38, PSet_LoLim := -1.5e+38, PSet_LoLoLim := -1.5e+38, MSet_SubstPV := 500.0, OSet_HiHiLim := 1.5e+38, OSet_HiLim := 1.5e+38, OSet_LoLim := -1.5e+38, OSet_LoLoLim := -1.5e+38, Set_SimPV := 500.0, Val := 500.0, Val_InpPV := 500.0, Val_PVEUMax := 20.0, Val_HiHiLim := 1.5e+38, Val_HiLim := 1.5e+38, Val_LoLim := -1.5e+38, Val_LoLoLim := -1.5e+38, Sts_InpPV := 1, Sts_PVBad := 1, Sts_Oper := 1, Sts_ProgOperLock := 1, Ack_HiHi := 1, Ack_Hi := 1, Ack_Lo := 1, Ack_LoLo := 1, Sts_Fail := 1, Ack_Fail := 1);   // From Secondary RAS To GBT Flow (FIT-600) 0-500 GPM
   SecRAS_ToGBT_Flow_Tot : U_FlowTot := (Inp_ProgStartReq := 1, Val_FlowRate := 500.0, Val_YearlyTot := 1.1457878);
   SolidsTk_Lv_Ain : P_AIn := (Inp_PV := 20.0, Cfg_SetTrack := 1, Cfg_PCmdClear := 1, Cfg_HasHiHiAlm := 1, Cfg_HasHiAlm := 1, Cfg_HasLoAlm := 1, Cfg_HasLoLoAlm := 1, Cfg_HiHiAckReqd := 1, Cfg_HiAckReqd := 1, Cfg_LoAckReqd := 1, Cfg_LoLoAckReqd := 1, Cfg_FailAckReqd := 1, Cfg_HiHiSeverity := 3, Cfg_HiSeverity := 2, Cfg_LoSeverity := 2, Cfg_LoLoSeverity := 3, Cfg_FailSeverity := 4, Cfg_InpRawMax := 20.0, Cfg_PVEUMax := 20.0, Cfg_HiHiDB := 1.0, Cfg_HiHiMinDuration := 5, Cfg_HiDB := 1.0, Cfg_HiMinDuration := 5, Cfg_LoDB := 1.0, Cfg_LoMinDuration := 5, Cfg_LoLoDB := 1.0, Cfg_LoLoMinDuration := 5, Cfg_FailHiLim := 45.0, Cfg_FailLoLim := -5.0, PSet_HiHiLim := 40.0, PSet_HiLim := 38.0, PSet_LoLim := 5.0, PSet_LoLoLim := 1.0, MSet_SubstPV := 20.0, OSet_HiHiLim := 40.0, OSet_HiLim := 38.0, OSet_LoLim := 5.0, OSet_LoLoLim := 1.0, Set_SimPV := 20.0, Val := 20.0, Val_InpPV := 20.0, Val_PVEUMax := 20.0, Val_HiHiLim := 40.0, Val_HiLim := 38.0, Val_LoLim := 5.0, Val_LoLoLim := 1.0, Sts_InpPV := 1, Sts_Oper := 1, Sts_ProgOperLock := 1, Ack_HiHi := 1, Ack_Hi := 1, Ack_Lo := 1, Ack_LoLo := 1, Ack_Fail := 1);   // Solids Storage Tank Level Indication (LIT-603) 0-20 Ft
   SolidsTkDrive_Intlk : P_Intlk := (Cfg_PCmdClear := 1, Sts_IntlkOK := 1, Sts_NBIntlkOK := 1);   // Solids Storage Tank #1 Drive Interlock
   SolidsTkDrive_Motor : P_Motor := (Inp_PermOK := 1, Inp_NBPermOK := 1, Inp_IntlkOK := 1, Inp_NBIntlkOK := 1, Inp_Sim := 1, Cfg_HasRunFdbk := 1, Cfg_UseRunFdbk := 1, Cfg_HasPermObj := 1, Cfg_HasIntlkObj := 1, Cfg_HasResInhObj := 1, Cfg_HasRunTimeObj := 1, Cfg_HasFailToStartAlm := 1, Cfg_HasFailToStopAlm := 1, Cfg_FailToStartAckReqd := 1, Cfg_FailToStopAckReqd := 1, Cfg_IntlkTripAckReqd := 1, Cfg_IOFaultAckReqd := 1, Cfg_FailToStartSeverity := 4, Cfg_FailToStopSeverity := 4, Cfg_IntlkTripSeverity := 2, Cfg_IOFaultSeverity := 4, Cfg_SimFdbkT := 2, Cfg_FailToStartT := 10, Cfg_FailToStopT := 10, PCmd_Acq := 1, Val_Notify := 1, Sts_Stopped := 1, Sts_Oper := 1, Sts_ProgOperLock := 1, Ack_FailToStop := 1, Ack_IntlkTrip := 1, Ack_IOFault := 1, Rdy_Start := 1, Rdy_Bypass := 1, Rdy_Disable := 1);   // Solids Storage Tank #1 Drive Motor
   SolidsTkDrive_Perm : P_Perm := (Inp_Perm00 := 1, Inp_Perm01 := 1, Inp_Perm02 := 1, Inp_Perm03 := 1, Inp_Perm04 := 1, Inp_Perm05 := 1, Inp_Perm06 := 1, Inp_Perm07 := 1, Inp_Perm08 := 1, Inp_Perm09 := 1, Inp_Perm10 := 1, Inp_Perm11 := 1, Inp_Perm12 := 1, Inp_Perm13 := 1, Inp_Perm14 := 1, Inp_Perm15 := 1, Sts_PermOK := 1, Sts_NBPermOK := 1, Sts_Perm := 2#1111_1111_1111_1111);   // Solids Storage Tank #1 Drive Permissive
   SolidsTkDrive_Reset : P_Reset := (Cfg_MinHoldTime := 1);   // Solids Storage Tank #1 Drive Reset
   SolidsTkDrive_ResInh : P_ResInh := (Inp_Stopped := 1, Cfg_ThreeColdStarts := 1800, Cfg_FirstFailCold := 1800, Cfg_SubseqFailCold := 14400, Cfg_FirstFailHot := 1800, Cfg_SubseqFailHot := 14400, Cfg_HotRestartOK := 3600, Cfg_RestartHot := 3600, Cfg_HotToCold := 57600, Val_State := 1, Sts_Ready := 1);   // Solids Storage Tank #1 Drive Restart Inhibit
   SolidsTkDrive_RunTime : P_RunTime := (Cfg_PCmdClear := 1, Val_Starts := 36, Val_CurRunHrs := 0.0010680555, Val_MaxRunHrs := 50.073418, Val_TotRunHrs := 50.4);   // Solids Storage Tank #1 Drive Run Time
   SolidsTkDrive_Torque : P_DIn := (Inp_Gate := 1, Cfg_NormTextVis := 1, Cfg_PCmdClear := 1, Cfg_TgtDisagreeAckReqd := 1, Cfg_TgtDisagreeSeverity := 3, Sts_InpPV := 1, Ack_TgtDisagree := 1, Rdy_SubstPV := 1);   // Solids Storage Tank #1 Drive Torque Fault
   WAS_HoldTkLv_Ain : P_AIn := (Cfg_SetTrack := 1, Cfg_PCmdClear := 1, Cfg_HasHiHiAlm := 1, Cfg_HasHiAlm := 1, Cfg_HasLoAlm := 1, Cfg_HasLoLoAlm := 1, Cfg_HiHiAckReqd := 1, Cfg_HiAckReqd := 1, Cfg_LoAckReqd := 1, Cfg_LoLoAckReqd := 1, Cfg_FailAckReqd := 1, Cfg_HiHiSeverity := 3, Cfg_HiSeverity := 2, Cfg_LoSeverity := 2, Cfg_LoLoSeverity := 3, Cfg_FailSeverity := 4, Cfg_InpRawMax := 20.0, Cfg_PVEUMax := 20.0, Cfg_HiHiDB := 1.0, Cfg_HiHiMinDuration := 5, Cfg_HiDB := 1.0, Cfg_HiMinDuration := 5, Cfg_LoDB := 1.0, Cfg_LoMinDuration := 5, Cfg_LoLoDB := 1.0, Cfg_LoLoMinDuration := 5, Cfg_FailHiLim := 1.5e+38, Cfg_FailLoLim := -1.5e+38, PSet_HiHiLim := 1.5e+38, PSet_HiLim := 1.5e+38, PSet_LoLim := -1.5e+38, PSet_LoLoLim := -1.5e+38, MSet_SubstPV := 10.0, OSet_HiHiLim := 1.5e+38, OSet_HiLim := 1.5e+38, OSet_LoLim := -1.5e+38, OSet_LoLoLim := -1.5e+38, Val := 10.0, Val_PVEUMax := 20.0, Val_HiHiLim := 1.5e+38, Val_HiLim := 1.5e+38, Val_LoLim := -1.5e+38, Val_LoLoLim := -1.5e+38, Sts_SubstPV := 1, Sts_Maint := 1, Ack_HiHi := 1, Ack_Hi := 1, Ack_Lo := 1, Ack_LoLo := 1, Ack_Fail := 1, Rdy_InpPV := 1);   // WAS Holding Tank Level Indication (LIT-608) 0-20 Ft
   WAS_StorageTkLv_Ain : P_AIn := (Inp_PV := 20.0, Cfg_SetTrack := 1, Cfg_PCmdClear := 1, Cfg_HasHiAlm := 1, Cfg_HasLoAlm := 1, Cfg_HiHiAckReqd := 1, Cfg_HiAckReqd := 1, Cfg_LoAckReqd := 1, Cfg_LoLoAckReqd := 1, Cfg_FailAckReqd := 1, Cfg_HiHiSeverity := 3, Cfg_HiSeverity := 2, Cfg_LoSeverity := 2, Cfg_LoLoSeverity := 3, Cfg_FailSeverity := 4, Cfg_InpRawMax := 40.0, Cfg_PVEUMax := 40.0, Cfg_HiHiDB := 1.0, Cfg_HiDB := 1.0, Cfg_HiMinDuration := 5, Cfg_LoDB := 1.0, Cfg_LoMinDuration := 5, Cfg_LoLoDB := 1.0, Cfg_FailHiLim := 45.0, Cfg_FailLoLim := -5.0, PSet_HiHiLim := 40.0, PSet_HiLim := 38.0, PSet_LoLim := 5.0, PSet_LoLoLim := 1.0, MSet_SubstPV := 20.0, OSet_HiHiLim := 40.0, OSet_HiLim := 38.0, OSet_LoLim := 5.0, OSet_LoLoLim := 1.0, Set_SimPV := 20.0, Val := 20.0, Val_InpPV := 20.0, Val_PVEUMax := 40.0, Val_HiHiLim := 40.0, Val_HiLim := 38.0, Val_LoLim := 5.0, Val_LoLoLim := 1.0, Sts_InpPV := 1, Sts_Oper := 1, Sts_ProgOperLock := 1, Ack_HiHi := 1, Ack_Hi := 1, Ack_Lo := 1, Ack_LoLo := 1, Ack_Fail := 1);   // WAS Storage Tank Level Indication (LIT-605) 0-20 Ft
END_VAR

PROGRAM MainProgram   (* main routine Main *)

ROUTINE A01_MiscDiscreteInputs   (* function block diagram *)
   SHEET 1
END_ROUTINE

ROUTINE A02_MiscAnalogInputs   (* function block diagram *)
   SHEET 1
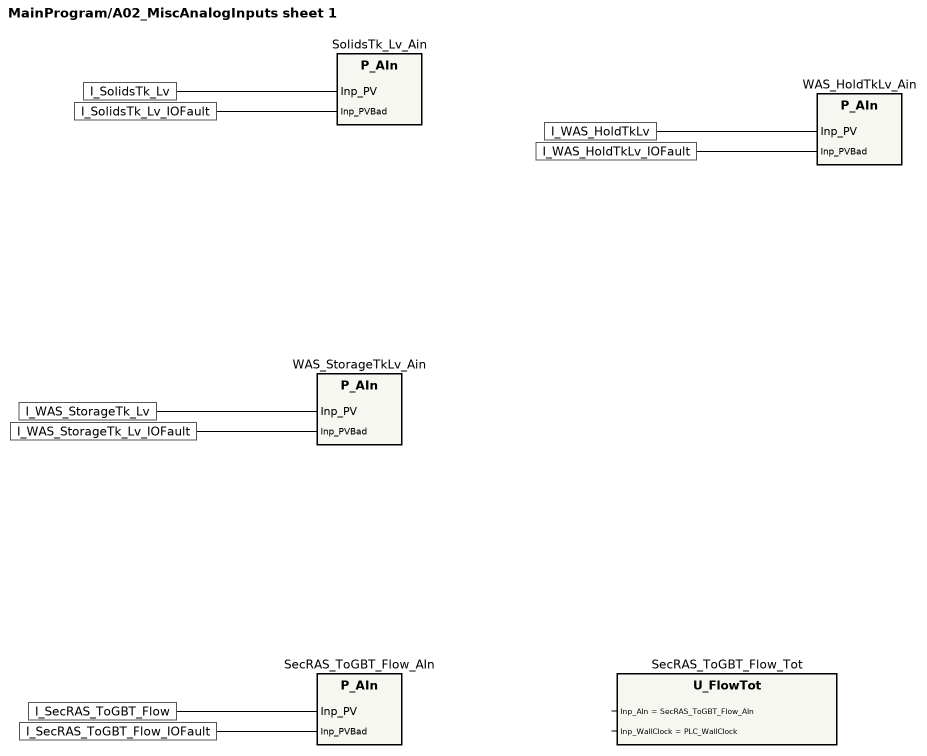
   WAS_StorageTkLv_Ain : P_AIn(Inp_PV := I_WAS_StorageTk_Lv, Inp_PVBad := I_WAS_StorageTk_Lv_IOFault);
   SecRAS_ToGBT_Flow_AIn : P_AIn(Inp_PV := I_SecRAS_ToGBT_Flow, Inp_PVBad := I_SecRAS_ToGBT_Flow_IOFault);
   SolidsTk_Lv_Ain : P_AIn(Inp_PV := I_SolidsTk_Lv, Inp_PVBad := I_SolidsTk_Lv_IOFault);
   SecRAS_ToGBT_Flow_Tot : U_FlowTot(Inp_AIn := SecRAS_ToGBT_Flow_AIn, Inp_WallClock := PLC_WallClock);
   WAS_HoldTkLv_Ain : P_AIn(Inp_PV := I_WAS_HoldTkLv, Inp_PVBad := I_WAS_HoldTkLv_IOFault);
END_ROUTINE

ROUTINE A03_MiscDiscreteOutputs   (* function block diagram *)
   SHEET 1
END_ROUTINE

ROUTINE A04_MiscAnalogOutputs   (* function block diagram *)
   SHEET 1
END_ROUTINE

ROUTINE Main   (* ladder *)
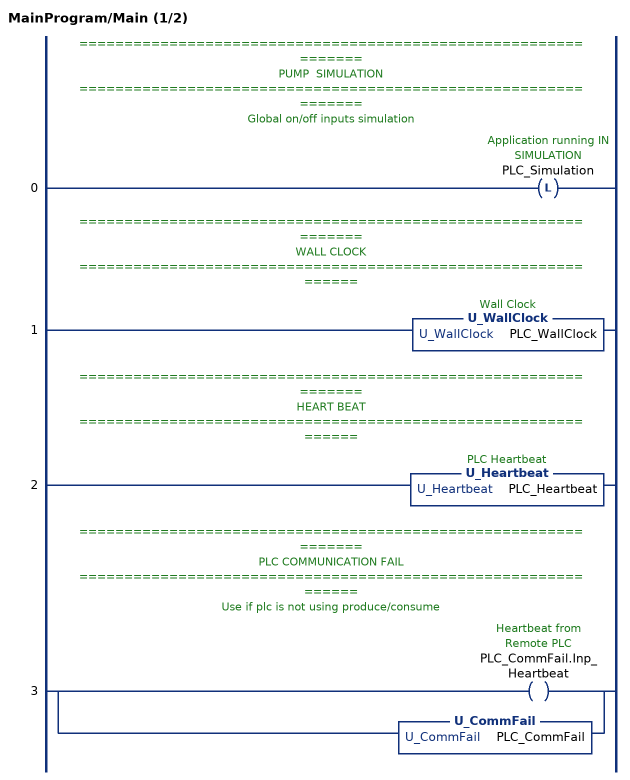
   // ===============================================================
   // PUMP  SIMULATION
   // ===============================================================
   // Global on/off inputs simulation
   0: OTL(PLC_Simulation);
   // ===============================================================
   // WALL CLOCK
   // ==============================================================
   1: U_WallClock(PLC_WallClock);
   // ===============================================================
   // HEART BEAT
   // ==============================================================
   2: U_Heartbeat(PLC_Heartbeat);
   // ===============================================================
   // PLC COMMUNICATION FAIL
   // ==============================================================
   // Use if plc is not using produce/consume
   3: [OTE(PLC_CommFail.Inp_Heartbeat) ,U_CommFail(PLC_CommFail) ];
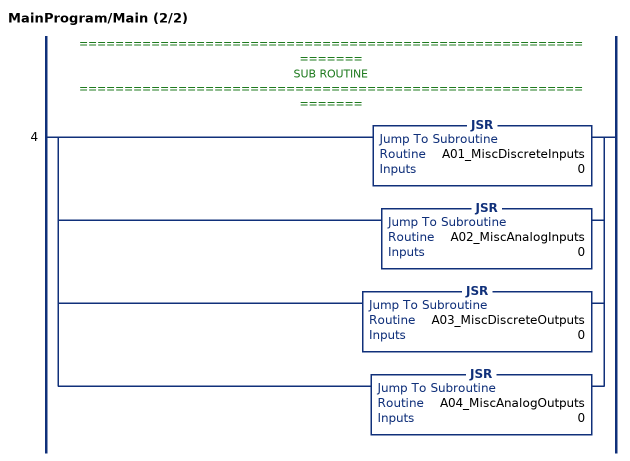
   // ===============================================================
   // SUB ROUTINE
   // ===============================================================
   4: [JSR(A01_MiscDiscreteInputs,0) ,JSR(A02_MiscAnalogInputs,0) ,JSR(A03_MiscDiscreteOutputs,0) ,JSR(A04_MiscAnalogOutputs,0) ];
END_ROUTINE
END_PROGRAM

PROGRAM PrimTkToSolidsTk01_Pump601   (* main routine Main *)
VAR
   Equip_Fault : ALIAS FOR I_P601_Fault;
   Equip_Fault_IOFault : ALIAS FOR I_P601_Fault_IOFault;
   Equip_GroupReset : ALIAS FOR PLC_Device_ResetPB;
   Equip_InAuto : ALIAS FOR I_P601_InAuto;
   Equip_InAuto_IOFault : ALIAS FOR I_P601_InAuto_IOFault;
   Equip_Intlk : ALIAS FOR P601_Intlk;
   Equip_IOFault : BOOL;
   Equip_Motor : ALIAS FOR P601_Motor;
   Equip_Out_Run : ALIAS FOR O_P601_Out_Run;
   Equip_RunFdbk : ALIAS FOR I_P601_RunFdbk;
   Equip_RunFdbk_IOFault : ALIAS FOR I_P601_RunFdbk_IOFault;
   Wrk_Hand : BOOL := 1;
   Wrk_ResetReqd : BOOL;
   Wrk_ResetRequired : BOOL;
END_VAR

ROUTINE A01_Pump_LDR   (* ladder *)
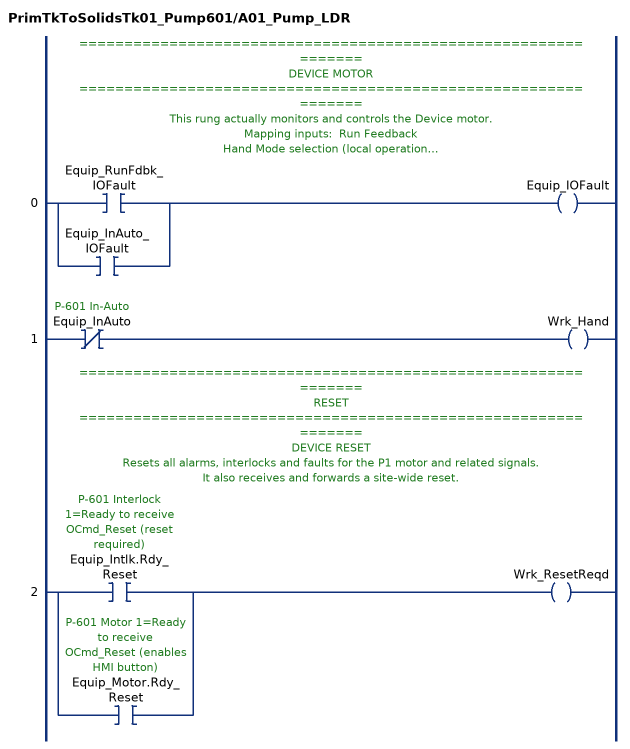
   // ===============================================================
   // DEVICE MOTOR
   // ===============================================================
   // This rung actually monitors and controls the Device motor.
   // Mapping inputs:  Run Feedback
   // Hand Mode selection (local operation)
   // Permissive OK
   // Protective’s OK,
   // I/O Fault signals
   // Pump Reset (above)
   // DEVICE
   // Output Mapping: Starter output
   0: [XIC(Equip_RunFdbk_IOFault) ,XIC(Equip_InAuto_IOFault) ]OTE(Equip_IOFault);
   1: XIO(Equip_InAuto)OTE(Wrk_Hand);
   // ===============================================================
   // RESET
   // ===============================================================
   // DEVICE RESET
   // Resets all alarms, interlocks and faults for the P1 motor and related signals.
   // It also receives and forwards a site-wide reset.
   2: [XIC(Equip_Intlk.Rdy_Reset) ,XIC(Equip_Motor.Rdy_Reset) ]OTE(Wrk_ResetReqd);
END_ROUTINE

ROUTINE A02_Pump_FBD   (* function block diagram *)
   SHEET 1   // Motor
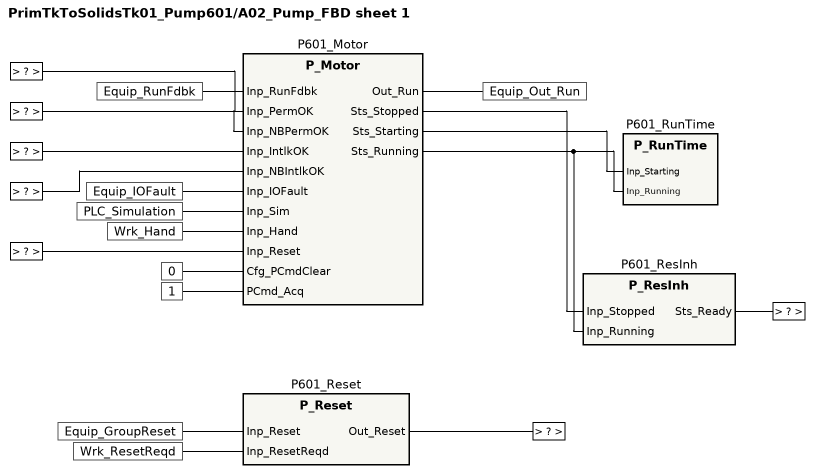
   P601_Reset : P_Reset(Inp_Reset := Equip_GroupReset, Inp_ResetReqd := Wrk_ResetReqd);
   WIRE(?) := P601_Reset.Out_Reset;
   P601_ResInh : P_ResInh(Inp_Stopped := P601_Motor.Sts_Stopped {feedback}, Inp_Running := P601_Motor.Sts_Running {feedback});
   WIRE(?) := P601_ResInh.Sts_Ready;
   P601_Motor : P_Motor(Inp_RunFdbk := Equip_RunFdbk, Inp_PermOK := WIRE(?), Inp_NBPermOK := WIRE(?), Inp_IntlkOK := WIRE(?), Inp_NBIntlkOK := WIRE(?), Inp_IOFault := Equip_IOFault, Inp_Sim := PLC_Simulation, Inp_Hand := Wrk_Hand, Inp_Reset := WIRE(?), Cfg_PCmdClear := 0, PCmd_Acq := 1);
   Equip_Out_Run := P601_Motor.Out_Run;
   P601_RunTime : P_RunTime(Inp_Starting := P601_Motor.Sts_Starting, Inp_Running := P601_Motor.Sts_Running);
   SHEET 2   // Permissives / Interlocks
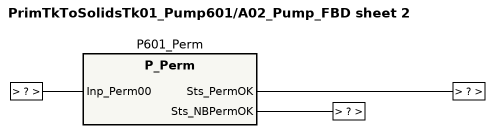
   P601_Perm : P_Perm(Inp_Perm00 := WIRE(?));
   WIRE(?) := P601_Perm.Sts_NBPermOK;
   WIRE(?) := P601_Perm.Sts_PermOK;
   SHEET 3   // Interlocks
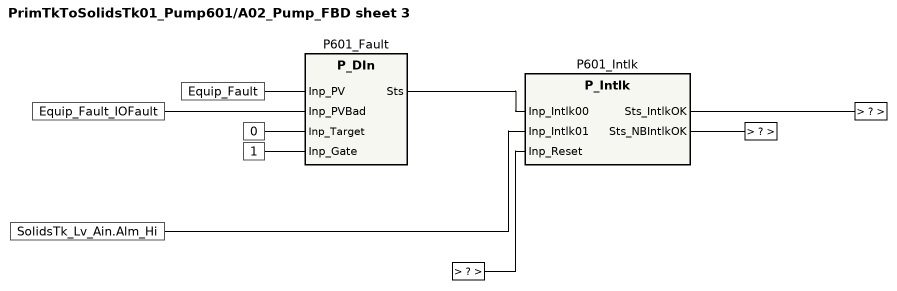
   P601_Fault : P_DIn(Inp_PV := Equip_Fault, Inp_PVBad := Equip_Fault_IOFault, Inp_Target := 0, Inp_Gate := 1);
   P601_Intlk : P_Intlk(Inp_Intlk00 := P601_Fault.Sts, Inp_Intlk01 := SolidsTk_Lv_Ain.Alm_Hi, Inp_Reset := WIRE(?));
   WIRE(?) := P601_Intlk.Sts_NBIntlkOK;
   WIRE(?) := P601_Intlk.Sts_IntlkOK;
END_ROUTINE

ROUTINE Main   (* ladder *)
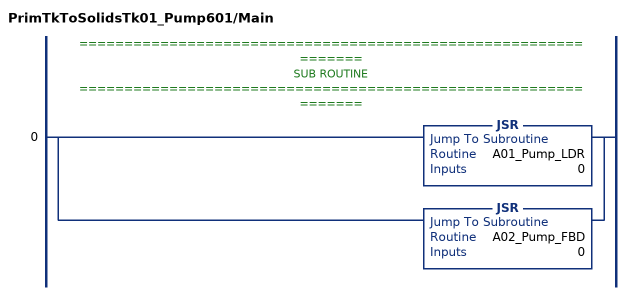
   // ===============================================================
   // SUB ROUTINE
   // ===============================================================
   0: [JSR(A01_Pump_LDR,0) ,JSR(A02_Pump_FBD,0) ];
END_ROUTINE
END_PROGRAM

PROGRAM SolidsTk01_Drive   (* main routine Main *)
VAR
   Equip_GroupReset : ALIAS FOR PLC_Device_ResetPB;
   Equip_InAuto : ALIAS FOR I_SolidsTkDrive_InAuto;
   Equip_InAuto_IOFault : ALIAS FOR I_SolidsTkDrive_InAuto_IOFault;
   Equip_Intlk : ALIAS FOR SolidsTkDrive_Intlk;
   Equip_IOFault : BOOL;
   Equip_Motor : ALIAS FOR SolidsTkDrive_Motor;
   Equip_Out_Run : ALIAS FOR O_SolidsTkDrive_Out_Run;
   Equip_RunFdbk : ALIAS FOR I_SolidsTkDrive_RunFdbk;
   Equip_RunFdbk_IOFault : ALIAS FOR I_SolidsTkDrive_RunFdbk_IOFault;
   Equip_Torque : ALIAS FOR I_SolidsTkDrive_Torque;
   Equip_Torque_IOFault : ALIAS FOR I_SolidsTkDrive_Torque_IOFault;
   Wrk_Hand : BOOL;
   Wrk_ResetReqd : BOOL;
   Wrk_ResetRequired : BOOL;
END_VAR

ROUTINE A01_Drive_LDR   (* ladder *)
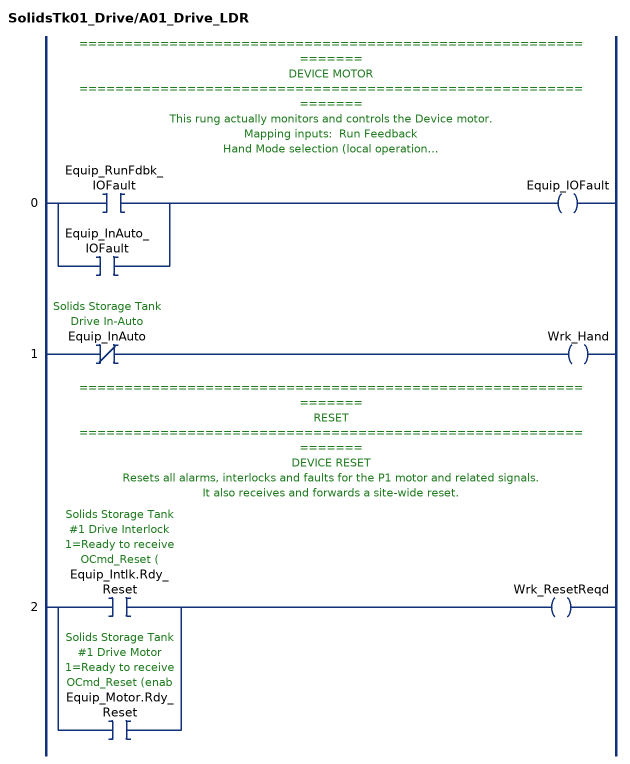
   // ===============================================================
   // DEVICE MOTOR
   // ===============================================================
   // This rung actually monitors and controls the Device motor.
   // Mapping inputs:  Run Feedback
   // Hand Mode selection (local operation)
   // Permissive OK
   // Protective’s OK,
   // I/O Fault signals
   // Pump Reset (above)
   // DEVICE
   // Output Mapping: Starter output
   0: [XIC(Equip_RunFdbk_IOFault) ,XIC(Equip_InAuto_IOFault) ]OTE(Equip_IOFault);
   1: XIO(Equip_InAuto)OTE(Wrk_Hand);
   // ===============================================================
   // RESET
   // ===============================================================
   // DEVICE RESET
   // Resets all alarms, interlocks and faults for the P1 motor and related signals.
   // It also receives and forwards a site-wide reset.
   2: [XIC(Equip_Intlk.Rdy_Reset) ,XIC(Equip_Motor.Rdy_Reset) ]OTE(Wrk_ResetReqd);
END_ROUTINE
